TYPE MyStruct :
STRUCT
	Par1 : INT;
	Par2 : INT;
END_STRUCT
END_TYPE

(* stored: Version 1.1.0.1, ProductVersion 3.1.4024.13
   DUT MyStruct: Id {61b03783-584a-4948-b581-2b1483ef01d0} *)
